// TIA Portal V18 export
DATA_BLOCK "heater status"   // DB141
{ S7_Optimized_Access := 'TRUE' }
VERSION : 0.1
// stored: AutoNumber true, DBAccessibleFromOPCUA true, IsOnlyStoredInLoadMemory false, IsRetainMemResEnabled false, IsWriteProtectedInAS false, MemoryReserve 100
   VAR
      temperature : Struct
         heater1 : Real;
         heater2 : Real;
         heater3 : Real;
         heater4 : Real;
      END_STRUCT;
   END_VAR
   VAR RETAIN
      "p100 connection okay" : Struct
         heater1 : Bool;
         heater2 : Bool;
         heater3 : Bool;
         heater4 : Bool;
      END_STRUCT;
   END_VAR
   VAR
      "Limit under temperature" : Struct
         heater1 : Bool;
         heater2 : Bool;
         heater3 : Bool;
         heater4 : Bool;
      END_STRUCT;
      "Limit Over temperature" : Struct
         heater1 : Bool;
         heater2 : Bool;
         heater3 : Bool;
         heater4 : Bool;
      END_STRUCT;
      "Dispensing Stop under temperature heater" { ExternalAccessible := 'False'; ExternalVisible := 'False'; ExternalWritable := 'False'} : Array[1..4] of Bool;
      "Critical Fault Stop Dispense Temperature NOK" : Bool;
      heater_nok : Bool;
   END_VAR
BEGIN
END_DATA_BLOCK
